              A_Touch_p[A_sel_v+9]=touch_4point(vr2_p1_up,vr2_p2_up,vr2_p3_up)
              $ 894 "A_Touch_p[A_sel_v+9]=ori_pose(A_Touch_p[A_sel_v+9],A_Touch_p[A_sel_v])"
              A_Touch_p[A_sel_v+9]=ori_pose(A_Touch_p[A_sel_v+9],A_Touch_p[A_sel_v])
            else:
              $ 895 "Else" "noBreak"
              $ 896 "If A_Touch_p[A_VR1]≟p[0,0,0,0,0,0]"
              if (A_Touch_p[A_VR1] == p[0,0,0,0,0,0]):
                $ 897 "Call MoveandTouchFun_3f"
                MoveandTouchFun_3f()
                $ 898 "touch_tmp≔A_Touch_p[A_sel_v]"
                global touch_tmp=A_Touch_p[A_sel_v]
                $ 899 "If A_Prepos_l[A_HOR_MR]≟p[0,0,0,0,0,0]"
                if (A_Prepos_l[A_HOR_MR] == p[0,0,0,0,0,0]):
                  $ 900 "direction(p[0,0,0,0,0,0],[0,1,0],8,120,160)"
                  direction(p[0,0,0,0,0,0],[0,1,0],8,120,160)
                  $ 901 "AAgcp≔get_actual_tcp_pose()"
                  global AAgcp= get_actual_tcp_pose ()
                  $ 902 "AAgangle≔up_right"
                  global AAgangle=p[.445203173045, -.406687378356, -.031125942276, 2.308490741423, -1.066468937023, 1.322151316133]
                  $ 903 "AAgtp≔p[AAgcp[0],AAgcp[1],AAgcp[2],AAgangle[3],AAgangle[4],AAgangle[5]]"
                  global AAgtp=p[AAgcp[0],AAgcp[1],AAgcp[2],AAgangle[3],AAgangle[4],AAgangle[5]]
                  $ 904 "MoveL"
                  $ 905 "AAgtp" "breakAfter"
                  movel(pose_trans(Base, AAgtp), a=0.08, v=0.08)
                  $ 907 "for_cal_zr≔contact_fun(p[0,0,0,0,0,0],[0,0,-1],20000,20,20)"
                  global for_cal_zr=contact_fun(p[0,0,0,0,0,0],[0,0,-1],20000,20,20)
                end
                $ 908 "touch_tmp[2]=for_cal_zr[2]"
                touch_tmp[2]=for_cal_zr[2]
                $ 909 "A_Touch_p[A_sel_v]=touch_tmp"
                A_Touch_p[A_sel_v]=touch_tmp
                $ 910 "for_cal_y_wel≔A_Touch_p[A_sel_v]"
                global for_cal_y_wel=A_Touch_p[A_sel_v]
                $ 911 "for_cal_x_wel≔A_Touch_p[A_sel_v]"
                global for_cal_x_wel=A_Touch_p[A_sel_v]
              else:
                $ 912 "Else" "noBreak"
                $ 913 "Call MoveFun"
                MoveFun()
                $ 914 "for_cal_y_wel≔contact_fun(p[0,0,0,0,0,0],[1,0,0],20000,20,20)"
                global for_cal_y_wel=contact_fun(p[0,0,0,0,0,0],[1,0,0],20000,20,20)
                $ 915 "direction(p[0,0,0,0,0,0],[-1,0,0],40,120,160)"
                direction(p[0,0,0,0,0,0],[-1,0,0],40,120,160)
                $ 916 "If A_Prepos_l[A_HOR_MR]≟p[0,0,0,0,0,0]"
                if (A_Prepos_l[A_HOR_MR] == p[0,0,0,0,0,0]):
                  $ 917 "direction(p[0,0,0,0,0,0],[0,-1,0],60,120,160)"
                  direction(p[0,0,0,0,0,0],[0,-1,0],60,120,160)
                  $ 918 "var_2≔contact_fun(p[0,0,0,0,0,0],[1,0,0],20000,20,20)"
                  global var_2=contact_fun(p[0,0,0,0,0,0],[1,0,0],20000,20,20)
                  $ 919 "direction(p[0,0,0,0,0,0],[-1,0,0],5,120,160)"
                  direction(p[0,0,0,0,0,0],[-1,0,0],5,120,160)
                  $ 920 "direction(p[0,0,0,0,0,0],[0,1,0],60,120,160)"
                  direction(p[0,0,0,0,0,0],[0,1,0],60,120,160)
                  $ 921 "direction(p[0,0,0,0,0,0],[1,0,0],10,120,160)"
                  direction(p[0,0,0,0,0,0],[1,0,0],10,120,160)
                  $ 922 "for_cal_x_wel≔contact_fun(p[0,0,0,0,0,0],[0,-1,0],20000,20,20)"
                  global for_cal_x_wel=contact_fun(p[0,0,0,0,0,0],[0,-1,0],20000,20,20)
                  $ 923 "direction(p[0,0,0,0,0,0],[0,1,0],20,120,160)"
                  direction(p[0,0,0,0,0,0],[0,1,0],20,120,160)
                  $ 924 "AAgcp≔get_actual_tcp_pose()"
                  global AAgcp= get_actual_tcp_pose ()
                  $ 925 "AAgangle≔up_right"
                  global AAgangle=p[.445203173045, -.406687378356, -.031125942276, 2.308490741423, -1.066468937023, 1.322151316133]
                  $ 926 "AAgtp≔p[AAgcp[0],AAgcp[1],AAgcp[2],AAgangle[3],AAgangle[4],AAgangle[5]]"
                  global AAgtp=p[AAgcp[0],AAgcp[1],AAgcp[2],AAgangle[3],AAgangle[4],AAgangle[5]]
                  $ 927 "MoveL"
                  $ 928 "AAgtp" "breakAfter"
                  movel(pose_trans(Base, AAgtp), a=0.1, v=0.1)
                  $ 930 "for_cal_zr≔contact_fun(p[0,0,0,0,0,0],[0,0,-1],20000,20,20)"
                  global for_cal_zr=contact_fun(p[0,0,0,0,0,0],[0,0,-1],20000,20,20)
                  $ 931 "direction(p[0,0,0,0,0,0],[0,0,1],20,120,160)"
                  direction(p[0,0,0,0,0,0],[0,0,1],20,120,160)
                  $ 932 "direction(p[0,0,0,0,0,0],[-1,0,0],20,120,160)"
                  direction(p[0,0,0,0,0,0],[-1,0,0],20,120,160)
                end
                $ 933 "for_cal_rot≔A_Touch_p[A_VR1]"
                global for_cal_rot=A_Touch_p[A_VR1]
                $ 934 "A_Touch_p[A_sel_v]=p[for_cal_y_wel[0],for_cal_x_wel[1],for_cal_zr[2],for_cal_rot[3],for_cal_rot[4],for_cal_rot[5]]"
                A_Touch_p[A_sel_v]=p[for_cal_y_wel[0],for_cal_x_wel[1],for_cal_zr[2],for_cal_rot[3],for_cal_rot[4],for_cal_rot[5]]
                $ 935 "write_welder(4, False )"
                write_welder(4,  False  )
              end
            end
            $ 936 "b2_par_cd≔0"
            global b2_par_cd=0
            $ 937 "homeing()"
            homeing()
          else:
            $ 938 "Else" "noBreak"
            $ 939 "homeing()"
            homeing()
          end
          $ 940 "write_welder(4,False)"
          write_welder(4,False)
          $ 997 "Touch After Offset"
          $ 998 "touch_after_offset"
          $ 999 "HOR"
          $ 1000 "If A_Prepos_l[A_HOR]≠p[0,0,0,0,0,0]"
          if (A_Prepos_l[A_HOR] != p[0,0,0,0,0,0]):
            $ 1001 "If b1_cell_info_L≟A or b1_cell_info_L≟C or b1_cell_info_L≟c"
            if (b1_cell_info_L == A  or  b1_cell_info_L == C  or  b1_cell_info_L == c):
              $ 1002 "If for_x_HOR≟p[0,0,0,0,0,0]"
              if (for_x_HOR == p[0,0,0,0,0,0]):
                $ 1003 "for_x_HOR≔A_Touch_p[A_VL1]"
                global for_x_HOR=A_Touch_p[A_VL1]
              end
              $ 1004 "If for_x_HOR≠p[0,0,0,0,0,0]"
              if (for_x_HOR != p[0,0,0,0,0,0]):
                $ 1005 "x_diff≔get_feature_pose(for_x_HOR,A_Touch_p[A_HOR])"
                global x_diff=get_feature_pose(for_x_HOR,A_Touch_p[A_HOR])
                $ 1006 "A_Touch_p[A_HOR]=pose_trans(A_Touch_p[A_HOR], p[x_diff[0],0,0,0,0,0])"
                A_Touch_p[A_HOR]= pose_trans (A_Touch_p[A_HOR], p[x_diff[0],0,0,0,0,0])
              end
            end
            $ 1007 "A_Touch_p[A_HOR]=pose_trans(A_Touch_p[A_HOR], p[offset_2f_begin/1000,0,0,0,0,0])"
            A_Touch_p[A_HOR]= pose_trans (A_Touch_p[A_HOR], p[offset_2f_begin/1000,0,0,0,0,0])
          end
          $ 1008 "VL1"
          $ 1009 "If A_Prepos_l[A_VL1]≠p[0,0,0,0,0,0]"
          if (A_Prepos_l[A_VL1] != p[0,0,0,0,0,0]):
            $ 1010 "If b1_cell_info_L≟A or b1_cell_info_L≟C or b1_cell_info_L≟c"
            if (b1_cell_info_L == A  or  b1_cell_info_L == C  or  b1_cell_info_L == c):
              $ 1011 "'3f only does not apply offset'"
              # '3f only does not apply offset'
              $ 1012 "If for_z_VL1≟p[0,0,0,0,0,0]"
              if (for_z_VL1 == p[0,0,0,0,0,0]):
                $ 1013 "for_z_VL1≔A_Touch_p[A_HOR]"
                global for_z_VL1=A_Touch_p[A_HOR]
              end
              $ 1014 "Comment"
              # Comment
              $ 1015 "If for_z_VL1≠p[0,0,0,0,0,0]"
              if (for_z_VL1 != p[0,0,0,0,0,0]):
                $ 1016 "z_diff≔get_feature_pose(for_z_VL1,A_Touch_p[A_VL1])"
                global z_diff=get_feature_pose(for_z_VL1,A_Touch_p[A_VL1])
                $ 1017 "A_Touch_p[A_VL1]=pose_trans(A_Touch_p[A_VL1], p[z_diff[0],0,0,0,0,0])"
                A_Touch_p[A_VL1]= pose_trans (A_Touch_p[A_VL1], p[z_diff[0],0,0,0,0,0])
              end
            end
            $ 1019 "A_Touch_p[A_VL1]=pose_trans(A_Touch_p[A_VL1], p[offset_3f_begin/1000,0,0,0,0,0])"
            A_Touch_p[A_VL1]= pose_trans (A_Touch_p[A_VL1], p[offset_3f_begin/1000,0,0,0,0,0])
          end
          $ 1020 "VL2"
          $ 1021 "If A_Prepos_l[A_VL2]≠p[0,0,0,0,0,0]"
          if (A_Prepos_l[A_VL2] != p[0,0,0,0,0,0]):
            $ 1022 "A_Touch_p[A_VL2]=pose_trans(A_Touch_p[A_VL2], p[offset_3f_begin/1000,0,0,0,0,0])"
            A_Touch_p[A_VL2]= pose_trans (A_Touch_p[A_VL2], p[offset_3f_begin/1000,0,0,0,0,0])
          end
          $ 1023 "HOR_R"
          $ 1024 "If A_Prepos_l[A_HOR_R]≠p[0,0,0,0,0,0]"
          if (A_Prepos_l[A_HOR_R] != p[0,0,0,0,0,0]):
            $ 1025 "If b1_cell_info_R≟A or b1_cell_info_R≟C or b1_cell_info_R≟c"
            if (b1_cell_info_R == A  or  b1_cell_info_R == C  or  b1_cell_info_R == c):
              $ 1026 "If for_x_HOR_R≟p[0,0,0,0,0,0]"
              if (for_x_HOR_R == p[0,0,0,0,0,0]):
                $ 1027 "for_x_HOR_R≔A_Touch_p[A_VR1]"
                global for_x_HOR_R=A_Touch_p[A_VR1]
              end
              $ 1028 "If for_x_HOR≠p[0,0,0,0,0,0]"
              if (for_x_HOR != p[0,0,0,0,0,0]):
                $ 1029 "x_diff≔get_feature_pose(for_x_HOR_R,A_Touch_p[A_HOR_R])"
                global x_diff=get_feature_pose(for_x_HOR_R,A_Touch_p[A_HOR_R])
                $ 1030 "A_Touch_p[A_HOR_R]=pose_trans(A_Touch_p[A_HOR_R], p[x_diff[0],0,0,0,0,0])"
                A_Touch_p[A_HOR_R]= pose_trans (A_Touch_p[A_HOR_R], p[x_diff[0],0,0,0,0,0])
              end
            end
            $ 1031 "A_Touch_p[A_HOR_R]=pose_trans(A_Touch_p[A_HOR_R], p[-offset_2f_begin/1000,0,0,0,0,0])"
            A_Touch_p[A_HOR_R]= pose_trans (A_Touch_p[A_HOR_R], p[-offset_2f_begin/1000,0,0,0,0,0])
          end
          $ 1032 "VR1"
          $ 1033 "If A_Prepos_l[A_VR1]≠p[0,0,0,0,0,0]"
          if (A_Prepos_l[A_VR1] != p[0,0,0,0,0,0]):
            $ 1034 "If b1_cell_info_R≟A or b1_cell_info_R≟C or b1_cell_info_R≟c"
            if (b1_cell_info_R == A  or  b1_cell_info_R == C  or  b1_cell_info_R == c):
              $ 1035 "If for_z_VR1≟p[0,0,0,0,0,0]"
              if (for_z_VR1 == p[0,0,0,0,0,0]):
                $ 1036 "for_z_VR1≔A_Touch_p[A_HOR_R]"
                global for_z_VR1=A_Touch_p[A_HOR_R]
              end
              $ 1037 "If for_z_VR1≠p[0,0,0,0,0,0]"
              if (for_z_VR1 != p[0,0,0,0,0,0]):
                $ 1038 "z_diff≔get_feature_pose(for_z_VR1,A_Touch_p[A_VR1])"
                global z_diff=get_feature_pose(for_z_VR1,A_Touch_p[A_VR1])
                $ 1039 "A_Touch_p[A_VR1]=pose_trans(A_Touch_p[A_VR1], p[z_diff[0],0,0,0,0,0])"
                A_Touch_p[A_VR1]= pose_trans (A_Touch_p[A_VR1], p[z_diff[0],0,0,0,0,0])
              end
            end
            $ 1041 "A_Touch_p[A_VR1]=pose_trans(A_Touch_p[A_VR1], p[offset_3f_begin/1000,0,0,0,0,0])"
            A_Touch_p[A_VR1]= pose_trans (A_Touch_p[A_VR1], p[offset_3f_begin/1000,0,0,0,0,0])
          end
          $ 1042 "VR2"
          $ 1043 "If A_Prepos_l[A_VR2]≠p[0,0,0,0,0,0]"
          if (A_Prepos_l[A_VR2] != p[0,0,0,0,0,0]):
            $ 1044 "A_Touch_p[A_VR2]=pose_trans(A_Touch_p[A_VR2], p[offset_3f_begin/1000,0,0,0,0,0])"
            A_Touch_p[A_VR2]= pose_trans (A_Touch_p[A_VR2], p[offset_3f_begin/1000,0,0,0,0,0])
          end
          $ 1045 "HOR_ML"
          $ 1046 "If A_Prepos_l[A_HOR_ML]≠p[0,0,0,0,0,0]"
          if (A_Prepos_l[A_HOR_ML] != p[0,0,0,0,0,0]):
            $ 1047 "A_Touch_p[A_HOR_M]=A_Touch_p[A_HOR_ML]"
            A_Touch_p[A_HOR_M]=A_Touch_p[A_HOR_ML]
            $ 1048 "x_welding_axis≔get_feature_pose(for_cal_x_wel,A_Touch_p[A_HOR_ML])"
            global x_welding_axis=get_feature_pose(for_cal_x_wel,A_Touch_p[A_HOR_ML])
            $ 1049 "A_Touch_p[A_HOR_M]=pose_trans(A_Touch_p[A_HOR_ML], p[x_welding_axis[0],0,0,0,0,0])"
            A_Touch_p[A_HOR_M]= pose_trans (A_Touch_p[A_HOR_ML], p[x_welding_axis[0],0,0,0,0,0])
            $ 1050 "A_Touch_p[A_HOR_M]=put_pose(A_Touch_p[A_HOR_M],0,for_cal_y_wel[0])"
            A_Touch_p[A_HOR_M]=put_pose(A_Touch_p[A_HOR_M],0,for_cal_y_wel[0])
            $ 1051 "A_Touch_p[A_HOR_M]=pose_trans(A_Touch_p[A_HOR_M], p[10/1000,0,0,0,0,0])"
            A_Touch_p[A_HOR_M]= pose_trans (A_Touch_p[A_HOR_M], p[10/1000,0,0,0,0,0])
            $ 1052 "If b1_cell_info_L≟C or b1_cell_info_L≟D"
            if (b1_cell_info_L == C  or  b1_cell_info_L == D):
              $ 1054 "x_welding_axis≔get_feature_pose(for_cal_x_wel,A_Touch_p[A_HOR_ML])"
              global x_welding_axis=get_feature_pose(for_cal_x_wel,A_Touch_p[A_HOR_ML])
              $ 1055 "A_Touch_p[A_HOR_ML]=pose_trans(A_Touch_p[A_HOR_ML],p[x_welding_axis[0],0,0,0,0,0])"
              A_Touch_p[A_HOR_ML]= pose_trans (A_Touch_p[A_HOR_ML],p[x_welding_axis[0],0,0,0,0,0])
              $ 1056 "A_Touch_p[A_HOR_ML]=pose_trans(A_Touch_p[A_HOR_ML],p[0/1000,0,0,0,0,0])"
              A_Touch_p[A_HOR_ML]= pose_trans (A_Touch_p[A_HOR_ML],p[0/1000,0,0,0,0,0])
            end
          end
          $ 1057 "HOR_MR"
          $ 1058 "If A_Prepos_l[A_HOR_MR]≠p[0,0,0,0,0,0]"
          if (A_Prepos_l[A_HOR_MR] != p[0,0,0,0,0,0]):
            $ 1060 "A_Touch_p[A_HOR_M]=A_Touch_p[A_HOR_MR]"
            A_Touch_p[A_HOR_M]=A_Touch_p[A_HOR_MR]
            $ 1061 "x_welding_axis≔get_feature_pose(for_cal_x_wel,A_Touch_p[A_HOR_MR])"
            global x_welding_axis=get_feature_pose(for_cal_x_wel,A_Touch_p[A_HOR_MR])
            $ 1062 "A_Touch_p[A_HOR_M]=pose_trans(A_Touch_p[A_HOR_M], p[x_welding_axis[0],0,0,0,0,0])"
            A_Touch_p[A_HOR_M]= pose_trans (A_Touch_p[A_HOR_M], p[x_welding_axis[0],0,0,0,0,0])
            $ 1063 "A_Touch_p[A_HOR_M]=put_pose(A_Touch_p[A_HOR_M],0,for_cal_y_wel[0])"
            A_Touch_p[A_HOR_M]=put_pose(A_Touch_p[A_HOR_M],0,for_cal_y_wel[0])
            $ 1064 "A_Touch_p[A_HOR_M]=pose_trans(A_Touch_p[A_HOR_M], p[-10/1000,0,0,0,0,0])"
            A_Touch_p[A_HOR_M]= pose_trans (A_Touch_p[A_HOR_M], p[-10/1000,0,0,0,0,0])
            $ 1065 "If b1_cell_info_R≟C or b1_cell_info_R≟D"
            if (b1_cell_info_R == C  or  b1_cell_info_R == D):
              $ 1067 "x_welding_axis≔get_feature_pose(for_cal_x_wel,A_Touch_p[A_HOR_MR])"
              global x_welding_axis=get_feature_pose(for_cal_x_wel,A_Touch_p[A_HOR_MR])
              $ 1068 "A_Touch_p[A_HOR_MR]=pose_trans(A_Touch_p[A_HOR_MR],p[x_welding_axis[0],0,0,0,0,0])"
              A_Touch_p[A_HOR_MR]= pose_trans (A_Touch_p[A_HOR_MR],p[x_welding_axis[0],0,0,0,0,0])
              $ 1069 "A_Touch_p[A_HOR_MR]=pose_trans(A_Touch_p[A_HOR_MR],p[-0/1000,0,0,0,0,0])"
              A_Touch_p[A_HOR_MR]= pose_trans (A_Touch_p[A_HOR_MR],p[-0/1000,0,0,0,0,0])
            end
          end
          $ 1070 "'Touch Remember On/OFF'"
          # 'Touch Remember On/OFF'
          $ 1071 "write_port_register(180,1)"
          write_port_register(180,1)
        else:
          $ 1072 "Else" "noBreak"
          $ 1073 "Ignore Touch and check error"
          $ 1074 "Auto_cur_cell≔0"
          global Auto_cur_cell=0
          $ 1075 "Loop Auto_cur_cell<Auto_total_cell"
          while (Auto_cur_cell<Auto_total_cell):
            $ 1076 "A_sel_v≔Auto_W_num[Auto_cur_cell]"
            global A_sel_v=Auto_W_num[Auto_cur_cell]
            $ 1077 "If A_sel_v<A_HOR_2path"
            if (A_sel_v<A_HOR_2path):
              $ 1078 "If A_Touch_p[A_sel_v]≟p[0,0,0,0,0,0]"
              if (A_Touch_p[A_sel_v] == p[0,0,0,0,0,0]):
                $ 1079 "write_port_register(142,120)"
                write_port_register(142,120)
                $ 1080 "Halt"
                halt
              end
            end
            $ 1081 "Auto_cur_cell≔Auto_cur_cell+1"
            global Auto_cur_cell=Auto_cur_cell+1
          end
          $ 1082 "Auto_cur_cell≔0"
          global Auto_cur_cell=0
        end
        $ 1083 "welding"
        $ 1084 "weldings"
        $ 1085 "Auto_cur_cell≔read_port_register(138)"
        global Auto_cur_cell= read_port_register (138)
        $ 1086 "time_cal_trig≔ True "
        global time_cal_trig=  True
        $ 1087 "Loop Auto_cur_cell<Auto_total_cell"
        while (Auto_cur_cell<Auto_total_cell):
          $ 1088 "write_port_register(138,Auto_cur_cell)"
          write_port_register(138,Auto_cur_cell)
          $ 1089 "running_trig≔ True "
          global running_trig=  True
          $ 1090 "'[2F_AB - 30] , [2F_CD_LEFT - 100] , [2F_CD_RIGHT - 150] , [3F - ELSE]'"
          # '[2F_AB - 30] , [2F_CD_LEFT - 100] , [2F_CD_RIGHT - 150] , [3F - ELSE]'
          $ 1091 "If Auto_W_num[Auto_cur_cell]≥100 and Auto_W_num[Auto_cur_cell]≤149"
          if (Auto_W_num[Auto_cur_cell] >= 100  and  Auto_W_num[Auto_cur_cell] <= 149):
            $ 1092 "'2F CD LEFT'"
            # '2F CD LEFT'
            $ 1093 "A_sel_v≔A_HOR"
            global A_sel_v=A_HOR
            $ 1094 "A_sel_v_end≔A_HOR_ML"
            global A_sel_v_end=A_HOR_ML
            $ 1095 "A_sel_v2≔A_HOR_M"
            global A_sel_v2=A_HOR_M
            $ 1096 "A_sel_v_end2≔A_HOR_R"
            global A_sel_v_end2=A_HOR_R
            $ 1097 "If floor(Auto_W_num[Auto_cur_cell]/10)≟10"
            if (floor(Auto_W_num[Auto_cur_cell]/10) == 10):
              $ 1098 "current_path≔1"
              global current_path=1
              $ 1099 "multi_path≔1"
              global multi_path=1
            else:
              $ 1100 "ElseIf floor(Auto_W_num[Auto_cur_cell]/10)≟11"
              if (floor(Auto_W_num[Auto_cur_cell]/10) == 11):
                $ 1101 "current_path≔2"
                global current_path=2
                $ 1102 "multi_path≔2"
                global multi_path=2
              else:
                $ 1103 "ElseIf floor(Auto_W_num[Auto_cur_cell]/10)≟12"
                if (floor(Auto_W_num[Auto_cur_cell]/10) == 12):
                  $ 1104 "current_path≔3"
                  global current_path=3
                  $ 1105 "multi_path≔3"
                  global multi_path=3
                else:
                  $ 1106 "ElseIf floor(Auto_W_num[Auto_cur_cell]/10)≟13"
                  if (floor(Auto_W_num[Auto_cur_cell]/10) == 13):
                    $ 1107 "current_path≔4"
                    global current_path=4
                    $ 1108 "multi_path≔4"
                    global multi_path=4
                  end
                end
              end
            end
            $ 1109 "current_2f≔current_2f+1"
            global current_2f=current_2f+1
            $ 1110 "CD_MLR≔ True "
            global CD_MLR=  True
            $ 1111 "write_port_register(135,A_HOR)"
            write_port_register(135,A_HOR)
            $ 1112 "write_port_register(136,current_2f)"
            write_port_register(136,current_2f)
            $ 1113 "If simulation_mode"
            if (simulation_mode):
              $ 1114 "Call welding_parameter_sim"
              welding_parameter_sim()
            else:
              $ 1115 "Else" "noBreak"
              $ 1116 "Call welding_parameter_init"
              welding_parameter_init()
            end
            $ 1117 "wv_direction≔1"
            global wv_direction=1
            $ 1118 "If Auto_W_num[Auto_cur_cell]%10≟4"
            if (Auto_W_num[Auto_cur_cell]%10 == 4):
              $ 1119 "A_sel_v≔A_HOR_R"
              global A_sel_v=A_HOR_R
              $ 1120 "Call MoveFun"
              MoveFun()
              $ 1121 "A_sel_v≔A_HOR"
              global A_sel_v=A_HOR
            else:
              $ 1122 "ElseIf Auto_W_num[Auto_cur_cell]%10≟0 or Auto_W_num[Auto_cur_cell]%10≟1 or Auto_W_num[Auto_cur_cell]%10≟2"
              if (Auto_W_num[Auto_cur_cell]%10 == 0  or  Auto_W_num[Auto_cur_cell]%10 == 1  or  Auto_W_num[Auto_cur_cell]%10 == 2):
                $ 1123 "Call MoveFun"
                MoveFun()
              end
            end
            $ 1124 "Call weav_welding_2f_CD"
            weav_welding_2f_CD()
          else:
            $ 1125 "ElseIf Auto_W_num[Auto_cur_cell]≥150 and Auto_W_num[Auto_cur_cell]≤189"
            if (Auto_W_num[Auto_cur_cell] >= 150  and  Auto_W_num[Auto_cur_cell] <= 189):
              $ 1126 "'2F CD RIGHT'"
              # '2F CD RIGHT'
              $ 1127 "A_sel_v≔A_HOR_R"
              global A_sel_v=A_HOR_R
              $ 1128 "A_sel_v_end≔A_HOR_MR"
              global A_sel_v_end=A_HOR_MR
              $ 1129 "A_sel_v2≔A_HOR_M"
              global A_sel_v2=A_HOR_M
              $ 1130 "A_sel_v_end2≔A_HOR"
              global A_sel_v_end2=A_HOR
              $ 1131 "If floor(Auto_W_num[Auto_cur_cell]/10)≟15"
              if (floor(Auto_W_num[Auto_cur_cell]/10) == 15):
                $ 1132 "current_path≔1"
                global current_path=1
                $ 1133 "multi_path≔1"
                global multi_path=1
              else:
                $ 1134 "ElseIf floor(Auto_W_num[Auto_cur_cell]/10)≟16"
                if (floor(Auto_W_num[Auto_cur_cell]/10) == 16):
                  $ 1135 "current_path≔2"
                  global current_path=2
                  $ 1136 "multi_path≔2"
                  global multi_path=2
                else:
                  $ 1137 "ElseIf floor(Auto_W_num[Auto_cur_cell]/10)≟17"
                  if (floor(Auto_W_num[Auto_cur_cell]/10) == 17):
                    $ 1138 "current_path≔3"
                    global current_path=3
                    $ 1139 "multi_path≔3"
                    global multi_path=3
                  else:
                    $ 1140 "ElseIf floor(Auto_W_num[Auto_cur_cell]/10)≟18"
                    if (floor(Auto_W_num[Auto_cur_cell]/10) == 18):
                      $ 1141 "current_path≔4"
                      global current_path=4
                      $ 1142 "multi_path≔4"
                      global multi_path=4
                    end
                  end
                end
              end
              $ 1143 "current_2f≔current_2f+1"
              global current_2f=current_2f+1
              $ 1144 "CD_MLR≔ False "
              global CD_MLR=  False
              $ 1145 "write_port_register(135,A_HOR)"
              write_port_register(135,A_HOR)
              $ 1146 "write_port_register(136,current_2f)"
              write_port_register(136,current_2f)
              $ 1147 "If simulation_mode"
              if (simulation_mode):
                $ 1148 "Call welding_parameter_sim"
                welding_parameter_sim()
              else:
                $ 1149 "Else" "noBreak"
                $ 1150 "Call welding_parameter_init"
                welding_parameter_init()
              end
              $ 1151 "wv_direction≔-1"
              global wv_direction=-1
              $ 1152 "If Auto_W_num[Auto_cur_cell]%10≟4"
              if (Auto_W_num[Auto_cur_cell]%10 == 4):
                $ 1153 "A_sel_v≔A_HOR"
                global A_sel_v=A_HOR
                $ 1154 "Call MoveFun"
                MoveFun()
                $ 1155 "A_sel_v≔A_HOR_R"
                global A_sel_v=A_HOR_R
              else:
                $ 1156 "ElseIf Auto_W_num[Auto_cur_cell]%10≟0 or Auto_W_num[Auto_cur_cell]%10≟1 or Auto_W_num[Auto_cur_cell]%10≟2"
                if (Auto_W_num[Auto_cur_cell]%10 == 0  or  Auto_W_num[Auto_cur_cell]%10 == 1  or  Auto_W_num[Auto_cur_cell]%10 == 2):
                  $ 1157 "Call MoveFun"
                  MoveFun()
                end
              end
              $ 1158 "Call weav_welding_2f_CD"
              weav_welding_2f_CD()
            else:
              $ 1159 "ElseIf Auto_W_num[Auto_cur_cell]≥30 and Auto_W_num[Auto_cur_cell]≤65"
              if (Auto_W_num[Auto_cur_cell] >= 30  and  Auto_W_num[Auto_cur_cell] <= 65):
                $ 1160 "'2F'"
                # '2F'
                $ 1161 "A_sel_v≔A_HOR"
                global A_sel_v=A_HOR
                $ 1162 "A_sel_v_end≔A_HOR_R"
                global A_sel_v_end=A_HOR_R
                $ 1163 "If floor(Auto_W_num[Auto_cur_cell]/10)≟3"
                if (floor(Auto_W_num[Auto_cur_cell]/10) == 3):
                  $ 1164 "current_path≔1"
                  global current_path=1
                  $ 1165 "multi_path≔1"
                  global multi_path=1
                else:
                  $ 1166 "ElseIf floor(Auto_W_num[Auto_cur_cell]/10)≟4"
                  if (floor(Auto_W_num[Auto_cur_cell]/10) == 4):
                    $ 1167 "current_path≔2"
                    global current_path=2
                    $ 1168 "multi_path≔2"
                    global multi_path=2
                  else:
                    $ 1169 "ElseIf floor(Auto_W_num[Auto_cur_cell]/10)≟5"
                    if (floor(Auto_W_num[Auto_cur_cell]/10) == 5):
                      $ 1170 "current_path≔3"
                      global current_path=3
                      $ 1171 "multi_path≔3"
                      global multi_path=3
                    else:
                      $ 1172 "ElseIf floor(Auto_W_num[Auto_cur_cell]/10)≟6"
                      if (floor(Auto_W_num[Auto_cur_cell]/10) == 6):
                        $ 1173 "current_path≔4"
                        global current_path=4
                        $ 1174 "multi_path≔4"
                        global multi_path=4
                      end
                    end
                  end
                end
                $ 1175 "current_2f≔current_2f+1"
                global current_2f=current_2f+1
                $ 1176 "write_port_register(135,A_HOR)"
                write_port_register(135,A_HOR)
                $ 1177 "write_port_register(136,current_2f)"
                write_port_register(136,current_2f)
                $ 1178 "If simulation_mode"
                if (simulation_mode):
                  $ 1179 "Call welding_parameter_sim"
                  welding_parameter_sim()
                else:
                  $ 1180 "Else" "noBreak"
                  $ 1181 "Call welding_parameter_init"
                  welding_parameter_init()
                end
                $ 1182 "If Auto_W_num[Auto_cur_cell]%10≟2"
                if (Auto_W_num[Auto_cur_cell]%10 == 2):
                  $ 1183 "A_sel_v≔A_HOR_R"
                  global A_sel_v=A_HOR_R
                  $ 1184 "Call MoveFun"
                  MoveFun()
                  $ 1185 "A_sel_v≔A_HOR"
                  global A_sel_v=A_HOR
                else:
                  $ 1186 "Else" "noBreak"
                  $ 1187 "Call MoveFun"
                  MoveFun()
                end
                $ 1188 "Call weav_welding_2f"
                weav_welding_2f()
              else:
                $ 1189 "Else" "noBreak"
                $ 1190 "A_sel_v≔Auto_W_num[Auto_cur_cell]"
                global A_sel_v=Auto_W_num[Auto_cur_cell]
                $ 1191 "write_port_register(135,A_sel_v)"
                write_port_register(135,A_sel_v)
                $ 1192 "current_path≔1"
                global current_path=1
                $ 1193 "current_2f≔0"
                global current_2f=0
                $ 1194 "write_port_register(136,current_2f)"
                write_port_register(136,current_2f)
                $ 1195 "If simulation_mode"
                if (simulation_mode):
                  $ 1196 "Call welding_parameter_sim"
                  welding_parameter_sim()
                else:
                  $ 1197 "Else" "noBreak"
                  $ 1198 "Call welding_parameter_init"
                  welding_parameter_init()
                end
                $ 1199 "A_sel_v_end≔A_sel_v+9"
                global A_sel_v_end=A_sel_v+9
                $ 1200 "Call weav_welding_3f"
                weav_welding_3f()
              end
            end
          end
          $ 1201 "Call reset_weld_param"
          reset_weld_param()
          $ 1204 "If get_move_trig≟1"
          if (get_move_trig == 1):
            $ 1205 "If get_next_number≠Auto_cur_cell"
            if (get_next_number != Auto_cur_cell):
              $ 1206 "Auto_cur_cell≔get_next_number"
              global Auto_cur_cell=get_next_number
            else:
              $ 1207 "Else" "noBreak"
              $ 1208 "Auto_cur_cell≔Auto_cur_cell+1"
              global Auto_cur_cell=Auto_cur_cell+1
            end
            $ 1209 "write_port_register(166,0)"
            write_port_register(166,0)
            $ 1210 "write_port_register(167,0)"
            write_port_register(167,0)
            $ 1211 "get_move_trig≔0"
            global get_move_trig=0
          else:
            $ 1212 "Else" "noBreak"
            $ 1213 "Auto_cur_cell≔Auto_cur_cell+1"
            global Auto_cur_cell=Auto_cur_cell+1
          end
        end
        $ 1214 "homeing()"
        homeing()
        $ 1215 "write_port_register(162,1)"
        write_port_register(162,1)
        $ 1216 "write_port_register(180,0)"
        write_port_register(180,0)
        thread_flag_304 = 1
      end
      if (a0_Job_Mode == 2):
        global thread_handler_304=run Thread_if_304()
        while (thread_flag_304 == 0):
          if not(a0_Job_Mode == 2):
            kill thread_handler_304
            thread_flag_304 = 2
          else:
            sync()
          end
        end
      else:
        thread_flag_304 = 2
      end
    end
    $ 1217 "Wait: 0.01"
    sleep(0.01)
    $ 1218 "after init auto"
    $ 1219 "If auto_on"
    if (auto_on):
      $ 1220 "write_port_register(202,0)"
      write_port_register(202,0)
      $ 1221 "timer_1: Stop"
      timer_1_is_counting = False
      $ 1222 "write_welder(0, False )"
      write_welder(0,  False  )
      $ 1223 "write_welder(4, False )"
      write_welder(4,  False  )
      $ 1224 "Call reset_weld_param"
      reset_weld_param()
      $ 1225 "multi_path≔1"
      global multi_path=1
      $ 1226 "auto_on≔ False "
      global auto_on=  False
      $ 1227 "current_2f≔0"
      global current_2f=0
      $ 1228 "get_center≔get_center_bak"
      global get_center=get_center_bak
      $ 1229 "vr2_p1≔p[0,0,0,0,0,0]"
      global vr2_p1=p[0,0,0,0,0,0]
      $ 1230 "welding_program≔ False "
      global welding_program=  False
      $ 1231 "start_num≔135"
      global start_num=135
      $ 1232 "Loop start_num<141"
      while (start_num<141):
        $ 1233 "write_port_register(start_num,0)"
        write_port_register(start_num,0)
        $ 1234 "start_num≔start_num+1"
        global start_num=start_num+1
      end
    end
  end
end
